SUBAPPLICATION Uebung_130_AX (* Übung zu ISOBUS Receive Message *)
  (* Standard: 61499-2; Description: Copyright (c) 2023 Meisterschulen am Ostbahnhof This program and the accompanying materials are made available under the terms of the Eclipse Public License 2.0 which is available at https://www.eclipse.org/legal/epl-2.0/ SPDX-License-Identifier: EPL-2.0 *)
  (* Version 1.0, 2023-10-23, Franz Höpfinger, Meisterschulen am Ostbahnhof, initial API and implementation and/or initial documentation *)
  PACKAGE Uebungen;
  IMPORT Uebungen::const::Uebung_120_129::Filter::PEAK_ADD;
  IMPORT Uebungen::const::Uebung_120_129::Filter::PEAK_FLT;
  IMPORT isobus::pgn::ISOUSERHOME_e::network;
  IMPORT isobus::pgn::ISO_CAN_NODE::NODE1;
  IMPORT isobus::pgn::const::PgnDef::PGN_PDU1_PropA;
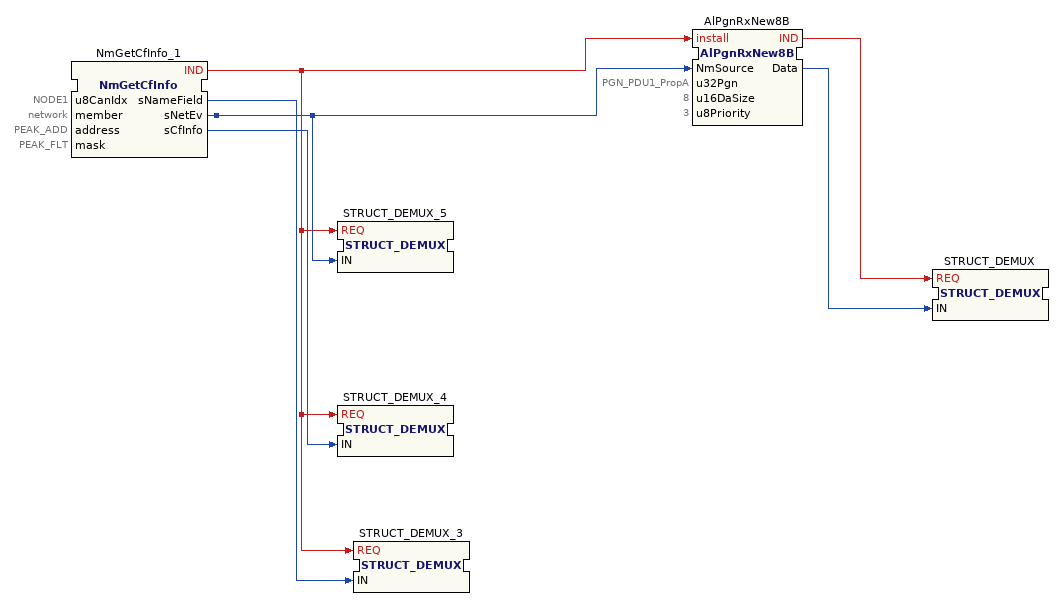
  FBS
    STRUCT_DEMUX_3 : eclipse4diac::convert::STRUCT_DEMUX; {SET_ATTRIBUTE(StructuredType, isobus::pgn::NAMEFIELD_T)}
    NmGetCfInfo_1 : isobus::pgn::NmGetCfInfo(u8CanIdx := NODE1, member := network, address := PEAK_ADD, mask := PEAK_FLT);
    STRUCT_DEMUX_4 : eclipse4diac::convert::STRUCT_DEMUX; {SET_ATTRIBUTE(StructuredType, isobus::pgn::CF_INFO_T)}
    STRUCT_DEMUX_5 : eclipse4diac::convert::STRUCT_DEMUX; {SET_ATTRIBUTE(StructuredType, isobus::pgn::ISONETEVENT_T)}
    AlPgnRxNew8B : isobus::pgn::rx::AlPgnRxNew8B(u32Pgn := PGN_PDU1_PropA, u16DaSize := 8, u8Priority := 3);
    STRUCT_DEMUX : eclipse4diac::convert::STRUCT_DEMUX; {SET_ATTRIBUTE(StructuredType, isobus::pgn::CAN_MSG)}
  END_FBS
  EVENT_CONNECTIONS
    NmGetCfInfo_1.IND TO STRUCT_DEMUX_3.REQ;
    NmGetCfInfo_1.IND TO STRUCT_DEMUX_4.REQ;
    NmGetCfInfo_1.IND TO STRUCT_DEMUX_5.REQ;
    NmGetCfInfo_1.IND TO AlPgnRxNew8B.install;
    AlPgnRxNew8B.IND TO STRUCT_DEMUX.REQ;
  END_CONNECTIONS
  DATA_CONNECTIONS
    NmGetCfInfo_1.sNameField TO STRUCT_DEMUX_3.IN;
    NmGetCfInfo_1.sNetEv TO STRUCT_DEMUX_5.IN;
    NmGetCfInfo_1.sCfInfo TO STRUCT_DEMUX_4.IN;
    NmGetCfInfo_1.sNetEv TO AlPgnRxNew8B.NmSource;
    AlPgnRxNew8B.Data TO STRUCT_DEMUX.IN;
  END_CONNECTIONS
END_SUBAPPLICATION
